FUNCTION_BLOCK RunUnitSlave EXTENDS RunUnitGeneric
VAR
	workingSignal : POINTER TO BOOL;  // start working when on
END_VAR

SUPER^();

CASE outputState OF 
	eSpecialStates.SLAVE_WORK_TRIGGER:
		//working start
		IF workingSignal^ THEN
			bWorkingOverride := TRUE; // backup working override signal
		END_IF
		IF bWorkingOverride AND NOT bIsBypassed THEN
			NextState := eSpecialStates.SLAVE_ENTER_PROCEDURE; // enter working procedure
		ELSIF bWorkingOverride AND bIsBypassed THEN
			NextState := eSpecialStates.SLAVE_WORK_DONE;
		ELSE
			//do nothing
		END_IF
	eSpecialStates.SLAVE_WORK_DONE:
		//working done
		workingSignal^ := FALSE;
		bWorkingOverride := FALSE;
		bMaterialOverride := FALSE;
		NextState := eSpecialStates.SLAVE_WORK_TRIGGER; // rewind
END_CASE

METHOD FB_init : BOOL
VAR_INPUT
	bInitRetains : BOOL; // if TRUE, the retain variables are initialized (warm start / cold start)
	bInCopyCode : BOOL;  // if TRUE, the instance afterwards gets moved into the copy code (online change)
	
	argParent : POINTER TO RunUnitGeneric;
	argSlotBase : POINTER TO RunMaterial;
	argSlotLast : POINTER TO RunMaterial;
	
	argWorkingSignal : POINTER TO BOOL;
END_VAR
//initialize 
Parent := argParent;
SlotBase := argSlotBase;
SlotLast := argSlotLast;
//
IF bInitRetains THEN
	NextState := eSpecialStates.INITIAL_BEGIN;
END_IF

workingSignal := argWorkingSignal; //link
END_METHOD

METHOD Initialize : BOOL
VAR_INPUT
END_VAR

IF State = eSpecialStates.INITIAL_END THEN
	//clear all internal status
	bEnStep := FALSE;
	bTrigStep := FALSE;
	bIsBypassed := FALSE;
	bWorkingOverride := FALSE;
	bMaterialOverride := FALSE;
	workingSignal^ := FALSE;	
END_IF
Initialize := SUPER^.Initialize();
END_METHOD

END_FUNCTION_BLOCK

(* stored: Version 1.1.0.1, ProductVersion 3.1.4022.10
   POU RunUnitSlave: Id {f294cd3d-3335-490a-8099-05ea45ee1c2b}, SpecialFunc None
   Method FB_init: Id {5fe09d05-6f33-419c-ac80-1bcb29fd85fb}
   Method Initialize: Id {d85590e7-7777-4ed2-a542-a41058c1988e} *)
